FUNCTION_BLOCK FB_TestFB

VAR
	nCounter : LINT;
END_VAR

nCounter : nCounter +1;

END_FUNCTION_BLOCK

(* stored: Version 1.1.0.1, ProductVersion 3.1.4024.9
   POU FB_TestFB: Id {5b834391-8053-4f7b-8fe8-f3aa3aadc7d8}, SpecialFunc None *)
